{attribute 'GeneratedUsingTerminal: EK1100-0000-0018'}
{attribute addProperty BoxType "EK1100-0000-0018"}
{attribute addProperty Id "Beckhoff_ER8xxxEK1122Beckhoff_ER8xxxEK1122_CCFAC45472"}
{attribute addProperty CRC "1352222121"}
{attribute addProperty Size "72"}
{attribute addProperty Name "Beckhoff ER8xxx"}
TYPE Beckhoff_ER8xxx_509945A9 EXTENDS EK1100_1FC0878B :
STRUCT
	{attribute addProperty Name "Beckhoff ER8xxxEK1122"}
	{attribute addProperty PreviousPort "Beckhoff ER8xxx : B"}
	Beckhoff_ER8xxxEK1122 : Beckhoff_ER8xxxEK1122_CCFAC454;
END_STRUCT
END_TYPE

(* stored: Version 1.2.0.0, ProductVersion 3.1.4024.11
   DUT Beckhoff_ER8xxx_509945A9: Id {2559b797-e2ab-4f37-a3c0-67467dc81644} *)
